// TIA Portal project "two-floor-elevator" (V20)

(* hardware
DEVICE "S7-1500/ET200MP-Station_1"  S7-1500 station
   slot 0: "Profilschiene_0"  Rack  6ES7 590-1***0-0AA0
   slot 1: "PLC_1"  CPU 1513-1 PN  6ES7 513-1AM03-0AB0  V4.0
      slot 3: "CPU-Display_1"  6ES7591-1AA00-0AA0
      slot 32768: "PROFINET-Schnittstelle_1"  X1
         slot 32769: "Port_1"  X1 P1
         slot 32770: "Port_2"  X1 P2
      slot 34817: "Virtual CP interface port_1"  Virtual CP interface port  Virtual CP interface port FW V4.0
   slot 2: "DI 16x24VDC BA_1"  DI 16x24VDC BA  6ES7 521-1BH10-0AA0  V1.1
   slot 3: "DQ 16x24VDC/0.5A ST_1"  DQ 16x24VDC/0.5A ST  6ES7 522-1BH00-0AB0  V2.0
   slot 4: "AI 8xU/I/R/RTD BA_1"  AI 8xU/I/R/RTD BA  6ES7 531-7QF00-0AB0  V1.0
   slot 5: "AQ 8xU/I HS_1"  AQ 8xU/I HS  6ES7 532-5HF00-0AB0  V2.2
*)

// ===== PLC "PLC_1"  CPU 1513-1 PN =====

VAR_GLOBAL   // PLC tag table "Standard-Variablentabelle"
   "PlcLabConnectIn01" AT %ID32760 : DWord;
   "PlcLabConnectIn02" AT %ID32764 : DWord;
   "PlcLabConnectOut01" AT %QD32760 : DWord;
   "PlcLabConnectOut02" AT %QD32764 : DWord;
END_VAR

VAR_GLOBAL   // PLC tag table "I/O"
   "Floor1Button" AT %I0.0 : Bool;   // Call/Go to Floor 1
   "Floor2Button" AT %I0.1 : Bool;   // Call/Go to Floor 2
   "Floor1Sensor" AT %I0.2 : Bool;   // Elevator is on Floor 1
   "Floor2Sensor" AT %I0.3 : Bool;   // Elevator is on Floor 2
   "EStop" AT %I0.5 : Bool;   // Emergency Stop the Elevator
   "MotorUp" AT %Q0.0 : Bool;   // Move Elevator Up
   "MotorDown" AT %Q0.1 : Bool;   // Move Elevator Down
   "Floor1Lamp" AT %Q0.3 : Bool;   // Floor 1 Indicator
   "Floor2Lamp" AT %Q0.4 : Bool;   // Floor 2 Indicator
END_VAR

ORGANIZATION_BLOCK "Main"   // OB1, LAD, ProgramCycle
TITLE = "Main Program Sweep (Cycle)"
{ S7_Optimized_Access := 'TRUE' }
VERSION : 0.1
   VAR_INPUT
      Initial_Call : Bool;   // Initial call of this OB
      Remanence : Bool;   // =True, if remanent data are available
   END_VAR
BEGIN

REGION Network 1: Move Elevator Up
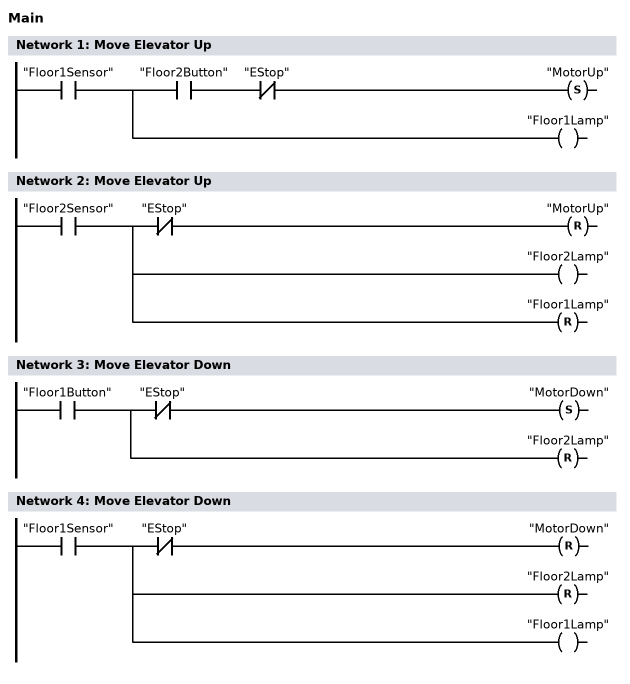
   RUNG wire#powerrail
      Contact( "Floor1Sensor" )
      wire#w1
      Contact( "Floor2Button" )
      I_Contact( "EStop" )
      S_Coil( "MotorUp" )
   END_RUNG
   RUNG wire#w1
      Coil( "Floor1Lamp" )
   END_RUNG
   // the same network as SCL:
   IF "Floor1Sensor" AND "Floor2Button" AND NOT "EStop" THEN "MotorUp" := TRUE; END_IF;
   "Floor1Lamp" := "Floor1Sensor";
END_REGION

REGION Network 2: Move Elevator Up
   RUNG wire#powerrail
      Contact( "Floor2Sensor" )
      wire#w1
      I_Contact( "EStop" )
      R_Coil( "MotorUp" )
   END_RUNG
   RUNG wire#w1
      Coil( "Floor2Lamp" )
   END_RUNG
   RUNG wire#w1
      R_Coil( "Floor1Lamp" )
   END_RUNG
   // the same network as SCL:
   IF "Floor2Sensor" AND NOT "EStop" THEN "MotorUp" := FALSE; END_IF;
   "Floor2Lamp" := "Floor2Sensor";
   IF "Floor2Sensor" THEN "Floor1Lamp" := FALSE; END_IF;
END_REGION

REGION Network 3: Move Elevator Down
   RUNG wire#powerrail
      Contact( "Floor1Button" )
      wire#w1
      I_Contact( "EStop" )
      S_Coil( "MotorDown" )
   END_RUNG
   RUNG wire#w1
      R_Coil( "Floor2Lamp" )
   END_RUNG
   // the same network as SCL:
   IF "Floor1Button" AND NOT "EStop" THEN "MotorDown" := TRUE; END_IF;
   IF "Floor1Button" THEN "Floor2Lamp" := FALSE; END_IF;
END_REGION

REGION Network 4: Move Elevator Down
   RUNG wire#powerrail
      Contact( "Floor1Sensor" )
      wire#w1
      I_Contact( "EStop" )
      R_Coil( "MotorDown" )
   END_RUNG
   RUNG wire#w1
      R_Coil( "Floor2Lamp" )
   END_RUNG
   RUNG wire#w1
      Coil( "Floor1Lamp" )
   END_RUNG
   // the same network as SCL:
   IF "Floor1Sensor" AND NOT "EStop" THEN "MotorDown" := FALSE; END_IF;
   IF "Floor1Sensor" THEN "Floor2Lamp" := FALSE; END_IF;
   "Floor1Lamp" := "Floor1Sensor";
END_REGION
END_ORGANIZATION_BLOCK